Staubli VAL3: listcreate.pgx

public program listCreate(string x_sTitle)
begin
  //-----------------------------------------------------------------------
  //Header begin
  //Description of program
  //  Create a list of data, displays the title x_sTitle,and draw
  //  the list from nTopX and nTopY position of the userPage (),
  //  of nBottomX length and height nListHeight.
  //
  //Input parameters
  //  string x_Title :
  //    role : Title that you want for the list of data
  //
  //Example
  //  Before using listCreate you can use setSizeList for defines all the
  //  parameters of position and size of the menu.
  //  call setSizeList(20,0,18,11)
  //  call listCreate("UserPage")
  //
  //History
  //  Creation : 28-04-08 - f.Rob
  //Header end
  //-----------------------------------------------------------------------
  sTitle=x_sTitle
  //Creation list of data
  call listFrame(sTitle,nTopX,nTopY,nBottomX,nListHeight)
  call listEmpty()
end
